// TIA Portal V20 export
TYPE "setTransferTimer"
// stored: Access Published, Namespace LineC1
   STRUCT
      setTransferTimer : Array[1..2] of Time;
   END_STRUCT;
END_TYPE
